PROGRAM pouMsgS1
VAR
	idbMsgAlarm: FB_CheckMessageBounds;
	idbMsgWarn: FB_CheckMessageBounds;
	idbMsgPrompt: FB_CheckMessageBounds;
END_VAR

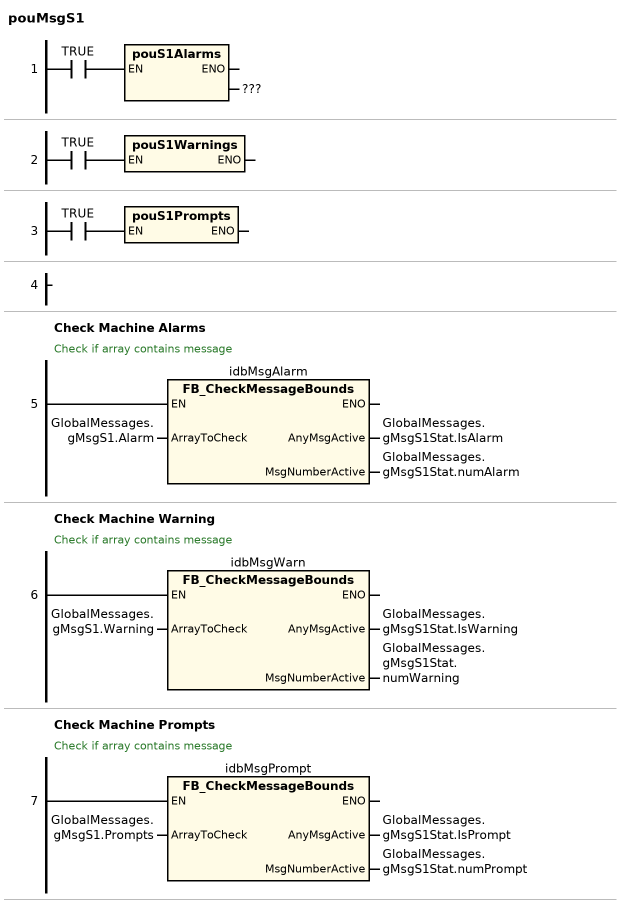
// NETWORK 1
pouS1Alarms();

// NETWORK 2
pouS1Warnings();

// NETWORK 3
pouS1Prompts();

// NETWORK 4

// NETWORK 5: Check Machine Alarms
// Check if array contains message
idbMsgAlarm(
    ArrayToCheck := GlobalMessages.gMsgS1.Alarm,
    AnyMsgActive => GlobalMessages.gMsgS1Stat.IsAlarm,
    MsgNumberActive => GlobalMessages.gMsgS1Stat.numAlarm); // FB_CheckMessageBounds

// NETWORK 6: Check Machine Warning
// Check if array contains message
idbMsgWarn(
    ArrayToCheck := GlobalMessages.gMsgS1.Warning,
    AnyMsgActive => GlobalMessages.gMsgS1Stat.IsWarning,
    MsgNumberActive => GlobalMessages.gMsgS1Stat.numWarning); // FB_CheckMessageBounds

// NETWORK 7: Check Machine Prompts
// Check if array contains message
idbMsgPrompt(
    ArrayToCheck := GlobalMessages.gMsgS1.Prompts,
    AnyMsgActive => GlobalMessages.gMsgS1Stat.IsPrompt,
    MsgNumberActive => GlobalMessages.gMsgS1Stat.numPrompt); // FB_CheckMessageBounds

END_PROGRAM

(* stored: Version 1.1.0.1, ProductVersion 3.1.4024.12
   POU pouMsgS1: Id {71043ed9-688e-4f83-bc07-eae8159a6d6f}, SpecialFunc None *)
